PROGRAM P_Prog1
VAR
	pDatePointer : POINTER TO DATE_AND_TIME := ADR(GVL.dtCurrentdate);
	nTimeRefrence : REFERENCE TO TIME := GVL.tTimeVar;
END_VAR

pDatePointer^ := DT#2023-02-08-15:31:19;
nTimeRefrence := T#2S;
GVL.aDateArray[2] := D#2023-02-25;
GVL.eSensor1 := E_SensorBrand.Bosch;
GVL.fbTimer(IN := GVL.bTimeStarter);
GVL.bOutQ := GVL.fbTimer.Q;
GVL.tElapseTime := GVL.fbTimer.ET;

END_PROGRAM

(* stored: Version 1.1.0.1, ProductVersion 3.1.4024.12
   POU P_Prog1: Id {6f86468e-f8b9-4717-87e3-d9e0af6e1dd8}, SpecialFunc None *)
